// TIA Portal project "pompaDzialajaca" (V15)

(* hardware
DEVICE "S7-1200 station_1"  S7-1200 Station
   slot 0: "Rack_0"  S7-1200 Rack  Rack  V1.0
   slot 1: "PLC_1"  CPU 1214C DC/DC/DC  6ES7 214-1AG40-0XB0  V4.2
      slot 3: "AQ 1x12BIT_1"  AQ1 signal board  6ES7 232-4HA30-0XB0  V1.0
   slot 101: "CM 1243-5"  CM 1243-5  6GK7 243-5DX30-0XE0  V1.3
   slot 102: "CM 1241 (RS485)_1"  CM 1241 (RS485)  6ES7 241-1CH30-0XB0  V1.0
*)

// ===== PLC "PLC_1"  CPU 1214C DC/DC/DC =====

VAR_GLOBAL   // PLC tag table "Default tag table"
   "start" AT %I0.0 : Bool;
   "poziomNiski" AT %Q0.1 : Bool;
   "stop" AT %I0.1 : Bool;
   "poziomWysoki" AT %Q0.3 : Bool;
   "CD" AT %I0.7 : Bool;
   "pompa" AT %Q1.0 : Bool;
   "awaria" AT %Q0.6 : Bool;
   "CG" AT %I0.6 : Bool;
   "sygAwaria" AT %Q0.7 : Bool;
   "poziomSredni" AT %Q0.2 : Bool;
   "Clock_Byte" AT %MB50 : Byte;
   "Clock_10Hz" AT %M50.0 : Bool;
   "Clock_5Hz" AT %M50.1 : Bool;
   "Clock_2.5Hz" AT %M50.2 : Bool;
   "Clock_2Hz" AT %M50.3 : Bool;
   "Clock_1.25Hz" AT %M50.4 : Bool;
   "Clock_1Hz" AT %M50.5 : Bool;
   "Clock_0.625Hz" AT %M50.6 : Bool;
   "Clock_0.5Hz" AT %M50.7 : Bool;
   "zboczeAwarii" AT %M12.0 : Bool;
   "pAwarii" AT %M14.0 : Bool;
END_VAR

ORGANIZATION_BLOCK "Main"   // OB1, LAD, ProgramCycle
TITLE = "Main Program Sweep (Cycle)"
{ S7_Optimized_Access := 'TRUE' }
VERSION : 0.1
   VAR_INPUT
      Initial_Call : Bool;   // Initial call of this OB
      Remanence : Bool;   // =True, if remanent data are available
   END_VAR
   VAR_TEMP   // added for the SCL form of the ladder/FBD networks
      _w1 : Bool;
   END_VAR
BEGIN

REGION Network 1
   // niski
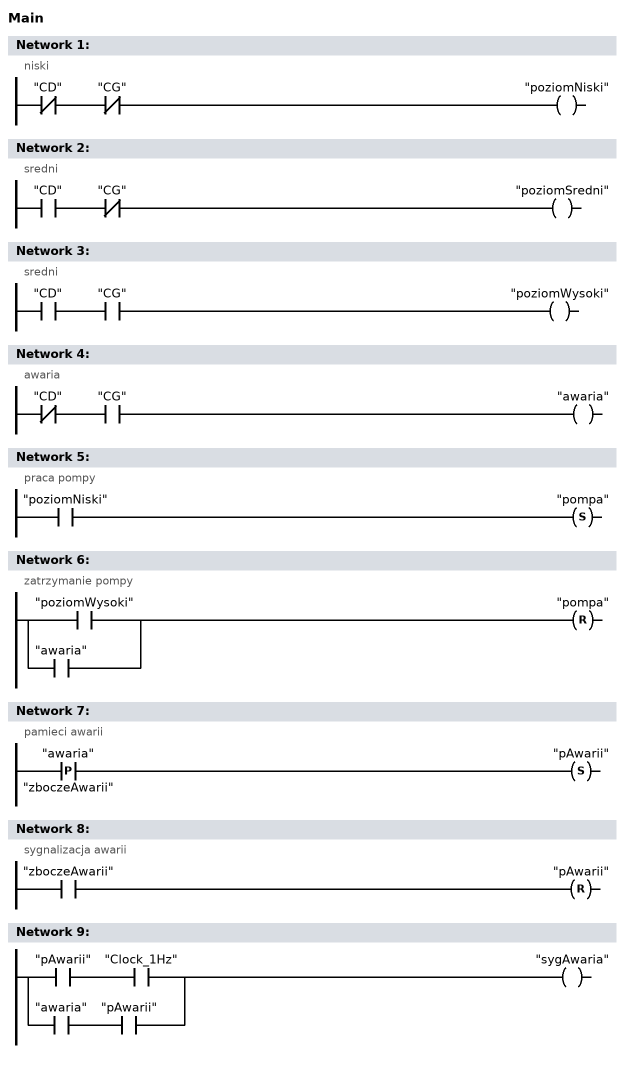
   RUNG wire#powerrail
      I_Contact( "CD" )
      I_Contact( "CG" )
      Coil( "poziomNiski" )
   END_RUNG
   // the same network as SCL:
   "poziomNiski" := NOT "CD" AND NOT "CG";
END_REGION

REGION Network 2
   // sredni
   RUNG wire#powerrail
      Contact( "CD" )
      I_Contact( "CG" )
      Coil( "poziomSredni" )
   END_RUNG
   // the same network as SCL:
   "poziomSredni" := "CD" AND NOT "CG";
END_REGION

REGION Network 3
   // sredni
   RUNG wire#powerrail
      Contact( "CD" )
      Contact( "CG" )
      Coil( "poziomWysoki" )
   END_RUNG
   // the same network as SCL:
   "poziomWysoki" := "CD" AND "CG";
END_REGION

REGION Network 4
   // awaria
   RUNG wire#powerrail
      I_Contact( "CD" )
      Contact( "CG" )
      Coil( "awaria" )
   END_RUNG
   // the same network as SCL:
   "awaria" := NOT "CD" AND "CG";
END_REGION

REGION Network 5
   // praca pompy
   RUNG wire#powerrail
      Contact( "poziomNiski" )
      S_Coil( "pompa" )
   END_RUNG
   // the same network as SCL:
   IF "poziomNiski" THEN "pompa" := TRUE; END_IF;
END_REGION

REGION Network 6
   // zatrzymanie pompy
   RUNG wire#powerrail
      Contact( "poziomWysoki" )
      wire#w1
      R_Coil( "pompa" )
   END_RUNG
   RUNG wire#powerrail
      Contact( "awaria" )
   END_RUNG wire#w1
   // the same network as SCL:
   IF "poziomWysoki" OR "awaria" THEN "pompa" := FALSE; END_IF;
END_REGION

REGION Network 7
   // pamieci awarii
   RUNG wire#powerrail
      P_Contact(operand := "awaria", bit := "zboczeAwarii")
      S_Coil( "pAwarii" )
   END_RUNG
   // the same network as SCL:
   #_w1 := "awaria" AND NOT "zboczeAwarii";   // rising edge of "awaria"
   "zboczeAwarii" := "awaria";
   IF #_w1 THEN "pAwarii" := TRUE; END_IF;
END_REGION

REGION Network 8
   // sygnalizacja awarii
   RUNG wire#powerrail
      Contact( "zboczeAwarii" )
      R_Coil( "pAwarii" )
   END_RUNG
   // the same network as SCL:
   IF "zboczeAwarii" THEN "pAwarii" := FALSE; END_IF;
END_REGION

REGION Network 9
   RUNG wire#powerrail
      Contact( "pAwarii" )
      Contact( "Clock_1Hz" )
      wire#w1
      Coil( "sygAwaria" )
   END_RUNG
   RUNG wire#powerrail
      Contact( "awaria" )
      Contact( "pAwarii" )
   END_RUNG wire#w1
   // the same network as SCL:
   "sygAwaria" := ("pAwarii" AND "Clock_1Hz") OR ("awaria" AND "pAwarii");
END_REGION
END_ORGANIZATION_BLOCK